FUNCTION_BLOCK Room_Ctx_Hmi
VAR_INPUT
	sStatusText				: Str;
	sErrorText				: Str;
	nStatusColor			: LWORD;
	
	bButton					: BOOL;
	sButtonText				: Str;
	nButtonColor			: LWORD;	
END_VAR
VAR_OUTPUT PERSISTENT
	rMaxPressure			: REAL := 2.0; // bar
	rMinPressure			: REAL := 0.2; // bar
	
	rMaxTemperature			: REAL := 65.0; // °C
	rStdTemperature			: REAL := 60.0; // °C
	rMinTemperature			: REAL := 55.0; // °C
END_VAR

END_FUNCTION_BLOCK

(* stored: Version 1.1.0.1
   POU Room_Ctx_Hmi: Id {9536c277-9786-455b-b876-b447754e1a8d}, SpecialFunc None *)
